VAR_GLOBAL CONSTANT
	cMAX_BLOCKED_SUP: INT := 3;
END_VAR

(* stored: Version 1.1.0.1, ProductVersion 3.1.0.23
   GVL Const_DRV: Id {bfc948d3-aed2-420b-b3ac-e40e075c9ae3} *)
